FUNCTION_BLOCK INTERNAL FB_DatabaseLoggerFactory EXTENDS FB_AbstractLoggerFactory
VAR
	pSQLServerLogger  : POINTER TO FB_SQLServerLogger;
    ipLogger          : ILogger := 0;
END_VAR

METHOD FB_exit : BOOL
VAR_INPUT
	bInCopyCode : BOOL; // if TRUE, the exit method is called for exiting an instance that is copied afterwards (online change).
END_VAR
IF (pSQLServerLogger <> 0) THEN
	__DELETE(pSQLServerLogger);
	pSQLServerLogger := 0;
END_IF
END_METHOD

METHOD FB_init : BOOL
VAR_INPUT
	bInitRetains : BOOL; // if TRUE, the retain variables are initialized (warm start / cold start)
	bInCopyCode  : BOOL;  // if TRUE, the instance afterwards gets moved into the copy code (online change)
	sDataSource  : STRING;
	sPassword    : STRING;
	sUser        : STRING;
END_VAR
pSQLServerLogger := __NEW(FB_SQLServerLogger);
ipLogger := pSQLServerLogger^;
END_METHOD

METHOD PUBLIC GetLogger : ILogger
VAR_INPUT
END_VAR
GetLogger := ipLogger;
END_METHOD

END_FUNCTION_BLOCK

(* stored: Version 1.1.0.1, ProductVersion 3.1.4024.12
   POU FB_DatabaseLoggerFactory: Id {369809d4-95c3-4440-8f66-e6799f12b2e0}, SpecialFunc None
   Method FB_exit: Id {14953acd-cc50-471a-b9fd-9dd9596a3671}
   Method FB_init: Id {27b68612-7ff3-495d-9528-2e92ddcc6785}
   Method GetLogger: Id {949a4117-b807-44c1-87ca-5ecbdbbb16e8} *)
